{attribute 'qualified_only'}
VAR_GLOBAL
	speed:					INT;
	target_speed:			INT;
	accelerating:			BOOL;
	braking:				BOOL;
	propulsion_fault: 		BOOL;
	propulsion_enable: 		BOOL;
	propulsion_active: 		BOOL;
	drive_voltages: INT;
END_VAR

(* stored: Version 1.1.0.1
   GVL GVL_Prop: Id {50abe306-50cd-40fe-9fcd-ded7060b0d4e} *)
